# EPICS autosave request: ipApp/Db/Oxford_CS800_settings.req
$(P)$(R)DEBUG
$(P)$(R)DISABLE
$(P)$(R)RRATE
$(P)$(R)RTEMP
$(P)$(R)PTIME
$(P)$(R)CTEMP
$(P)$(R)ERATE
